TYPE PuckLnSwAction :
STRUCT

	OkTo_ReleasePuck: BOOL;
	OkTo_Fault: BOOL;
	Target_Workstop: cLaneSel;
	Target_Lane: cLaneSel;
	Target_FaultCode: DINT;
	Target_PuckLnSw: PuckLnSw; //Used for Debug and Visualization

END_STRUCT
END_TYPE

(* stored: Version 1.1.0.1, ProductVersion 3.1.4024.6
   DUT PuckLnSwAction: Id {502e032a-13cd-43a3-b23d-dc0dcc1704dc} *)
